// TwinCAT 3 PLC project SaftyPLC
// ProgramVersion: 3.1.4026.13
// libraries:
//   Tc2_Standard, * (Beckhoff Automation GmbH)
//   Tc2_System, * (Beckhoff Automation GmbH)
//   Tc3_Module, * (Beckhoff Automation GmbH)
// project tree:
//   GVLs/ GVL_Safety.TcGVL
//   / PlcTask.TcTTO
//   POUs/ MAIN.TcPOU
// (motion and I/O tree: see PLC project planartrackmovement)
// real-time tasks:
//   TASK XTS Task: cycle T#500us, priority 1, ADS port 350
//   TASK Job Task: cycle default, priority 32
//   TASK MC-Task (MET): cycle T#2ms, priority 3, ADS port 521
//   TASK MC-Task (MPT): cycle T#10ms, priority 8, ADS port 531
//   TASK PlcTask: cycle T#2ms, priority 20, ADS port 351
// variable links:
//   SaftyPLC/SaftyPLC Instance <-> Device 1 (EtherCAT)/Term 1 (EK1200)/Term 13 (EL2912)
//     PlcTask Inputs/GVL_Safety.SaeftyOk <-> StandardInputs/TwinSafeGroup1.SafetyOk_72
//     PlcTask Inputs/GVL_Safety.SafetyInRun <-> StandardInputs/TwinSafeGroup1.SafetyInRun_73
//     PlcTask Outputs/GVL_Safety.Reset <-> StandardOutputs/TwinSafeGroup1.ErrorAcknowledgement_1
//     PlcTask Outputs/GVL_Safety.Run <-> StandardOutputs/TwinSafeGroup1.Run_2
//     PlcTask Outputs/GVL_Safety.Start <-> StandardOutputs/TwinSafeGroup1.STO_75
//   SaftyPLC/SaftyPLC Instance <-> Device 1 (EtherCAT)/Term 1 (EK1200)/Term 2 (EL1809)
//     PlcTask Inputs/GVL_Safety.HWReset <-> Channel 16/Input
//     PlcTask Inputs/GVL_Safety.HWStart <-> Channel 14/Input
//     PlcTask Inputs/GVL_Safety.HWStop <-> Channel 15/Input
//   SaftyPLC/SaftyPLC Instance <-> Device 1 (EtherCAT)/Term 1 (EK1200)/Term 4 (EL2809)
//     PlcTask Outputs/MAIN.xRequestReset <-> Channel 16/Output
//   SaftyPLC/SaftyPLC Instance <-> Device 4 (EtherCAT)/Box 50 (AT5100-0100)
//     PlcTask Outputs/GVL_Safety.Reset <-> Module 1 (SAFETY)/SAFETY Standard Outputdata/Standard In Var 1
//     PlcTask Outputs/GVL_Safety.Run <-> Module 1 (SAFETY)/SAFETY Standard Outputdata/Standard In Var 2
//   SaftyPLC/SaftyPLC Instance <-> Device 4 (EtherCAT)/Box 51 (AT5100-0100)
//     PlcTask Outputs/GVL_Safety.Reset <-> Module 1 (SAFETY)/SAFETY Standard Outputdata/Standard In Var 1
//     PlcTask Outputs/GVL_Safety.Run <-> Module 1 (SAFETY)/SAFETY Standard Outputdata/Standard In Var 2
//   SaftyPLC/SaftyPLC Instance <-> Device 4 (EtherCAT)/Box 52 (AT5100-0100)
//     PlcTask Outputs/GVL_Safety.Reset <-> Module 1 (SAFETY)/SAFETY Standard Outputdata/Standard In Var 1
//     PlcTask Outputs/GVL_Safety.Run <-> Module 1 (SAFETY)/SAFETY Standard Outputdata/Standard In Var 2
//   SaftyPLC/SaftyPLC Instance <-> Device 4 (EtherCAT)/Box 53 (AT5100-0100)
//     PlcTask Outputs/GVL_Safety.Reset <-> Module 1 (SAFETY)/SAFETY Standard Outputdata/Standard In Var 1
//     PlcTask Outputs/GVL_Safety.Run <-> Module 1 (SAFETY)/SAFETY Standard Outputdata/Standard In Var 2
//   SaftyPLC/SaftyPLC Instance <-> Device 4 (EtherCAT)/Box 54 (AT5100-0100)
//     PlcTask Outputs/GVL_Safety.Reset <-> Module 1 (SAFETY)/SAFETY Standard Outputdata/Standard In Var 1
//     PlcTask Outputs/GVL_Safety.Run <-> Module 1 (SAFETY)/SAFETY Standard Outputdata/Standard In Var 2
//   SaftyPLC/SaftyPLC Instance <-> Device 4 (EtherCAT)/Box 55 (AT5100-0100)
//     PlcTask Outputs/GVL_Safety.Reset <-> Module 1 (SAFETY)/SAFETY Standard Outputdata/Standard In Var 1
//     PlcTask Outputs/GVL_Safety.Run <-> Module 1 (SAFETY)/SAFETY Standard Outputdata/Standard In Var 2
//   SaftyPLC/SaftyPLC Instance <-> Device 4 (EtherCAT)/Box 56 (AT5100-0100)
//     PlcTask Outputs/GVL_Safety.Reset <-> Module 1 (SAFETY)/SAFETY Standard Outputdata/Standard In Var 1
//     PlcTask Outputs/GVL_Safety.Run <-> Module 1 (SAFETY)/SAFETY Standard Outputdata/Standard In Var 2
//   SaftyPLC/SaftyPLC Instance <-> Device 4 (EtherCAT)/Box 57 (AT5100-0100)
//     PlcTask Outputs/GVL_Safety.Reset <-> Module 1 (SAFETY)/SAFETY Standard Outputdata/Standard In Var 1
//     PlcTask Outputs/GVL_Safety.Run <-> Module 1 (SAFETY)/SAFETY Standard Outputdata/Standard In Var 2
//   SaftyPLC/SaftyPLC Instance <-> Device 4 (EtherCAT)/Box 58 (AT5100-0100)
//     PlcTask Outputs/GVL_Safety.Reset <-> Module 1 (SAFETY)/SAFETY Standard Outputdata/Standard In Var 1
//     PlcTask Outputs/GVL_Safety.Run <-> Module 1 (SAFETY)/SAFETY Standard Outputdata/Standard In Var 2
//   SaftyPLC/SaftyPLC Instance <-> Device 4 (EtherCAT)/Box 59 (AT5100-0100)
//     PlcTask Outputs/GVL_Safety.Reset <-> Module 1 (SAFETY)/SAFETY Standard Outputdata/Standard In Var 1
//     PlcTask Outputs/GVL_Safety.Run <-> Module 1 (SAFETY)/SAFETY Standard Outputdata/Standard In Var 2
//   SaftyPLC/SaftyPLC Instance <-> Device 4 (EtherCAT)/Box 60 (AT5100-0100)
//     PlcTask Outputs/GVL_Safety.Reset <-> Module 1 (SAFETY)/SAFETY Standard Outputdata/Standard In Var 1
//     PlcTask Outputs/GVL_Safety.Run <-> Module 1 (SAFETY)/SAFETY Standard Outputdata/Standard In Var 2
//   SaftyPLC/SaftyPLC Instance <-> Device 4 (EtherCAT)/Box 61 (AT5100-0100)
//     PlcTask Outputs/GVL_Safety.Reset <-> Module 1 (SAFETY)/SAFETY Standard Outputdata/Standard In Var 1
//     PlcTask Outputs/GVL_Safety.Run <-> Module 1 (SAFETY)/SAFETY Standard Outputdata/Standard In Var 2
//   SaftyPLC/SaftyPLC Instance <-> Device 4 (EtherCAT)/Box 62 (AT5100-0100)
//     PlcTask Outputs/GVL_Safety.Reset <-> Module 1 (SAFETY)/SAFETY Standard Outputdata/Standard In Var 1
//     PlcTask Outputs/GVL_Safety.Run <-> Module 1 (SAFETY)/SAFETY Standard Outputdata/Standard In Var 2
//   SaftyPLC/SaftyPLC Instance <-> Device 4 (EtherCAT)/Box 63 (AT5100-0100)
//     PlcTask Outputs/GVL_Safety.Reset <-> Module 1 (SAFETY)/SAFETY Standard Outputdata/Standard In Var 1
//     PlcTask Outputs/GVL_Safety.Run <-> Module 1 (SAFETY)/SAFETY Standard Outputdata/Standard In Var 2
//   SaftyPLC/SaftyPLC Instance <-> Device 4 (EtherCAT)/Box 64 (AT5100-0100)
//     PlcTask Outputs/GVL_Safety.Reset <-> Module 1 (SAFETY)/SAFETY Standard Outputdata/Standard In Var 1
//     PlcTask Outputs/GVL_Safety.Run <-> Module 1 (SAFETY)/SAFETY Standard Outputdata/Standard In Var 2
//   SaftyPLC/SaftyPLC Instance <-> Device 4 (EtherCAT)/Box 65 (AT5100-0100)
//     PlcTask Outputs/GVL_Safety.Reset <-> Module 1 (SAFETY)/SAFETY Standard Outputdata/Standard In Var 1
//     PlcTask Outputs/GVL_Safety.Run <-> Module 1 (SAFETY)/SAFETY Standard Outputdata/Standard In Var 2
//   SaftyPLC/SaftyPLC Instance <-> Device 4 (EtherCAT)/Box 66 (AT5100-0100)
//     PlcTask Outputs/GVL_Safety.Reset <-> Module 1 (SAFETY)/SAFETY Standard Outputdata/Standard In Var 1
//     PlcTask Outputs/GVL_Safety.Run <-> Module 1 (SAFETY)/SAFETY Standard Outputdata/Standard In Var 2
//   SaftyPLC/SaftyPLC Instance <-> Device 4 (EtherCAT)/Box 67 (AT5100-0100)
//     PlcTask Outputs/GVL_Safety.Reset <-> Module 1 (SAFETY)/SAFETY Standard Outputdata/Standard In Var 1
//     PlcTask Outputs/GVL_Safety.Run <-> Module 1 (SAFETY)/SAFETY Standard Outputdata/Standard In Var 2
//   SaftyPLC/SaftyPLC Instance <-> Device 4 (EtherCAT)/Box 68 (AT5100-0100)
//     PlcTask Outputs/GVL_Safety.Reset <-> Module 1 (SAFETY)/SAFETY Standard Outputdata/Standard In Var 1
//     PlcTask Outputs/GVL_Safety.Run <-> Module 1 (SAFETY)/SAFETY Standard Outputdata/Standard In Var 2
//   SaftyPLC/SaftyPLC Instance <-> Device 4 (EtherCAT)/Box 69 (AT5100-0100)
//     PlcTask Outputs/GVL_Safety.Reset <-> Module 1 (SAFETY)/SAFETY Standard Outputdata/Standard In Var 1
//     PlcTask Outputs/GVL_Safety.Run <-> Module 1 (SAFETY)/SAFETY Standard Outputdata/Standard In Var 2
//   SaftyPLC/SaftyPLC Instance <-> Device 4 (EtherCAT)/Box 70 (AT5100-0100)
//     PlcTask Outputs/GVL_Safety.Reset <-> Module 1 (SAFETY)/SAFETY Standard Outputdata/Standard In Var 1
//     PlcTask Outputs/GVL_Safety.Run <-> Module 1 (SAFETY)/SAFETY Standard Outputdata/Standard In Var 2
//   SaftyPLC/SaftyPLC Instance <-> Device 4 (EtherCAT)/Box 71 (AT5100-0100)
//     PlcTask Outputs/GVL_Safety.Reset <-> Module 1 (SAFETY)/SAFETY Standard Outputdata/Standard In Var 1
//     PlcTask Outputs/GVL_Safety.Run <-> Module 1 (SAFETY)/SAFETY Standard Outputdata/Standard In Var 2
//   SaftyPLC/SaftyPLC Instance <-> Device 4 (EtherCAT)/Box 72 (AT5100-0100)
//     PlcTask Outputs/GVL_Safety.Reset <-> Module 1 (SAFETY)/SAFETY Standard Outputdata/Standard In Var 1
//     PlcTask Outputs/GVL_Safety.Run <-> Module 1 (SAFETY)/SAFETY Standard Outputdata/Standard In Var 2
//   SaftyPLC/SaftyPLC Instance <-> Device 4 (EtherCAT)/Box 73 (AT5100-0100)
//     PlcTask Outputs/GVL_Safety.Reset <-> Module 1 (SAFETY)/SAFETY Standard Outputdata/Standard In Var 1
//     PlcTask Outputs/GVL_Safety.Run <-> Module 1 (SAFETY)/SAFETY Standard Outputdata/Standard In Var 2
//   SaftyPLC/SaftyPLC Instance <-> Device 4 (EtherCAT)/Box 74 (AT5100-0100)
//     PlcTask Outputs/GVL_Safety.Reset <-> Module 1 (SAFETY)/SAFETY Standard Outputdata/Standard In Var 1
//     PlcTask Outputs/GVL_Safety.Run <-> Module 1 (SAFETY)/SAFETY Standard Outputdata/Standard In Var 2
//   SaftyPLC/SaftyPLC Instance <-> Device 4 (EtherCAT)/Box 75 (AT5100-0100)
//     PlcTask Outputs/GVL_Safety.Reset <-> Module 1 (SAFETY)/SAFETY Standard Outputdata/Standard In Var 1
//     PlcTask Outputs/GVL_Safety.Run <-> Module 1 (SAFETY)/SAFETY Standard Outputdata/Standard In Var 2
//   SaftyPLC/SaftyPLC Instance <-> Device 4 (EtherCAT)/Box 76 (AT5100-0100)
//     PlcTask Outputs/GVL_Safety.Reset <-> Module 1 (SAFETY)/SAFETY Standard Outputdata/Standard In Var 1
//     PlcTask Outputs/GVL_Safety.Run <-> Module 1 (SAFETY)/SAFETY Standard Outputdata/Standard In Var 2
//   SaftyPLC/SaftyPLC Instance <-> Device 4 (EtherCAT)/Box 77 (AT5100-0100)
//     PlcTask Outputs/GVL_Safety.Reset <-> Module 1 (SAFETY)/SAFETY Standard Outputdata/Standard In Var 1
//     PlcTask Outputs/GVL_Safety.Run <-> Module 1 (SAFETY)/SAFETY Standard Outputdata/Standard In Var 2
//   SaftyPLC/SaftyPLC Instance <-> Device 4 (EtherCAT)/Box 78 (AT5100-0100)
//     PlcTask Outputs/GVL_Safety.Reset <-> Module 1 (SAFETY)/SAFETY Standard Outputdata/Standard In Var 1
//     PlcTask Outputs/GVL_Safety.Run <-> Module 1 (SAFETY)/SAFETY Standard Outputdata/Standard In Var 2
//   SaftyPLC/SaftyPLC Instance <-> Device 4 (EtherCAT)/Box 79 (AT5100-0100)
//     PlcTask Outputs/GVL_Safety.Reset <-> Module 1 (SAFETY)/SAFETY Standard Outputdata/Standard In Var 1
//     PlcTask Outputs/GVL_Safety.Run <-> Module 1 (SAFETY)/SAFETY Standard Outputdata/Standard In Var 2
//   SaftyPLC/SaftyPLC Instance <-> Device 4 (EtherCAT)/Box 80 (AT5100-0100)
//     PlcTask Outputs/GVL_Safety.Reset <-> Module 1 (SAFETY)/SAFETY Standard Outputdata/Standard In Var 1
//     PlcTask Outputs/GVL_Safety.Run <-> Module 1 (SAFETY)/SAFETY Standard Outputdata/Standard In Var 2
//   SaftyPLC/SaftyPLC Instance <-> Device 4 (EtherCAT)/Box 81 (AT5100-0100)
//     PlcTask Outputs/GVL_Safety.Reset <-> Module 1 (SAFETY)/SAFETY Standard Outputdata/Standard In Var 1
//     PlcTask Outputs/GVL_Safety.Run <-> Module 1 (SAFETY)/SAFETY Standard Outputdata/Standard In Var 2
//   SaftyPLC/SaftyPLC Instance <-> Device 8 (EtherCAT)/Box 18 (AT5100-0100)
//     PlcTask Outputs/GVL_Safety.Reset <-> Module 1 (SAFETY)/SAFETY Standard Outputdata/Standard In Var 1
//     PlcTask Outputs/GVL_Safety.Run <-> Module 1 (SAFETY)/SAFETY Standard Outputdata/Standard In Var 2
//   SaftyPLC/SaftyPLC Instance <-> Device 8 (EtherCAT)/Box 19 (AT5100-0100)
//     PlcTask Outputs/GVL_Safety.Reset <-> Module 1 (SAFETY)/SAFETY Standard Outputdata/Standard In Var 1
//     PlcTask Outputs/GVL_Safety.Run <-> Module 1 (SAFETY)/SAFETY Standard Outputdata/Standard In Var 2
//   SaftyPLC/SaftyPLC Instance <-> Device 8 (EtherCAT)/Box 20 (AT5100-0100)
//     PlcTask Outputs/GVL_Safety.Reset <-> Module 1 (SAFETY)/SAFETY Standard Outputdata/Standard In Var 1
//     PlcTask Outputs/GVL_Safety.Run <-> Module 1 (SAFETY)/SAFETY Standard Outputdata/Standard In Var 2
//   SaftyPLC/SaftyPLC Instance <-> Device 8 (EtherCAT)/Box 21 (AT5100-0100)
//     PlcTask Outputs/GVL_Safety.Reset <-> Module 1 (SAFETY)/SAFETY Standard Outputdata/Standard In Var 1
//     PlcTask Outputs/GVL_Safety.Run <-> Module 1 (SAFETY)/SAFETY Standard Outputdata/Standard In Var 2
//   SaftyPLC/SaftyPLC Instance <-> Device 8 (EtherCAT)/Box 22 (AT5100-0100)
//     PlcTask Outputs/GVL_Safety.Reset <-> Module 1 (SAFETY)/SAFETY Standard Outputdata/Standard In Var 1
//     PlcTask Outputs/GVL_Safety.Run <-> Module 1 (SAFETY)/SAFETY Standard Outputdata/Standard In Var 2
//   SaftyPLC/SaftyPLC Instance <-> Device 8 (EtherCAT)/Box 23 (AT5100-0100)
//     PlcTask Outputs/GVL_Safety.Reset <-> Module 1 (SAFETY)/SAFETY Standard Outputdata/Standard In Var 1
//     PlcTask Outputs/GVL_Safety.Run <-> Module 1 (SAFETY)/SAFETY Standard Outputdata/Standard In Var 2
//   SaftyPLC/SaftyPLC Instance <-> Device 8 (EtherCAT)/Box 24 (AT5100-0100)
//     PlcTask Outputs/GVL_Safety.Reset <-> Module 1 (SAFETY)/SAFETY Standard Outputdata/Standard In Var 1
//     PlcTask Outputs/GVL_Safety.Run <-> Module 1 (SAFETY)/SAFETY Standard Outputdata/Standard In Var 2
//   SaftyPLC/SaftyPLC Instance <-> Device 8 (EtherCAT)/Box 25 (AT5100-0100)
//     PlcTask Outputs/GVL_Safety.Reset <-> Module 1 (SAFETY)/SAFETY Standard Outputdata/Standard In Var 1
//     PlcTask Outputs/GVL_Safety.Run <-> Module 1 (SAFETY)/SAFETY Standard Outputdata/Standard In Var 2
//   SaftyPLC/SaftyPLC Instance <-> Device 8 (EtherCAT)/Box 26 (AT5100-0100)
//     PlcTask Outputs/GVL_Safety.Reset <-> Module 1 (SAFETY)/SAFETY Standard Outputdata/Standard In Var 1
//     PlcTask Outputs/GVL_Safety.Run <-> Module 1 (SAFETY)/SAFETY Standard Outputdata/Standard In Var 2
//   SaftyPLC/SaftyPLC Instance <-> Device 8 (EtherCAT)/Box 27 (AT5100-0100)
//     PlcTask Outputs/GVL_Safety.Reset <-> Module 1 (SAFETY)/SAFETY Standard Outputdata/Standard In Var 1
//     PlcTask Outputs/GVL_Safety.Run <-> Module 1 (SAFETY)/SAFETY Standard Outputdata/Standard In Var 2
//   SaftyPLC/SaftyPLC Instance <-> Device 8 (EtherCAT)/Box 28 (AT5100-0100)
//     PlcTask Outputs/GVL_Safety.Reset <-> Module 1 (SAFETY)/SAFETY Standard Outputdata/Standard In Var 1
//     PlcTask Outputs/GVL_Safety.Run <-> Module 1 (SAFETY)/SAFETY Standard Outputdata/Standard In Var 2
//   SaftyPLC/SaftyPLC Instance <-> Device 8 (EtherCAT)/Box 29 (AT5100-0100)
//     PlcTask Outputs/GVL_Safety.Reset <-> Module 1 (SAFETY)/SAFETY Standard Outputdata/Standard In Var 1
//     PlcTask Outputs/GVL_Safety.Run <-> Module 1 (SAFETY)/SAFETY Standard Outputdata/Standard In Var 2
//   SaftyPLC/SaftyPLC Instance <-> Device 8 (EtherCAT)/Box 30 (AT5100-0100)
//     PlcTask Outputs/GVL_Safety.Reset <-> Module 1 (SAFETY)/SAFETY Standard Outputdata/Standard In Var 1
//     PlcTask Outputs/GVL_Safety.Run <-> Module 1 (SAFETY)/SAFETY Standard Outputdata/Standard In Var 2
//   SaftyPLC/SaftyPLC Instance <-> Device 8 (EtherCAT)/Box 31 (AT5100-0100)
//     PlcTask Outputs/GVL_Safety.Reset <-> Module 1 (SAFETY)/SAFETY Standard Outputdata/Standard In Var 1
//     PlcTask Outputs/GVL_Safety.Run <-> Module 1 (SAFETY)/SAFETY Standard Outputdata/Standard In Var 2
//   SaftyPLC/SaftyPLC Instance <-> Device 8 (EtherCAT)/Box 32 (AT5100-0100)
//     PlcTask Outputs/GVL_Safety.Reset <-> Module 1 (SAFETY)/SAFETY Standard Outputdata/Standard In Var 1
//     PlcTask Outputs/GVL_Safety.Run <-> Module 1 (SAFETY)/SAFETY Standard Outputdata/Standard In Var 2
//   SaftyPLC/SaftyPLC Instance <-> Device 8 (EtherCAT)/Box 33 (AT5100-0100)
//     PlcTask Outputs/GVL_Safety.Reset <-> Module 1 (SAFETY)/SAFETY Standard Outputdata/Standard In Var 1
//     PlcTask Outputs/GVL_Safety.Run <-> Module 1 (SAFETY)/SAFETY Standard Outputdata/Standard In Var 2
//   SaftyPLC/SaftyPLC Instance <-> Device 8 (EtherCAT)/Box 34 (AT5100-0100)
//     PlcTask Outputs/GVL_Safety.Reset <-> Module 1 (SAFETY)/SAFETY Standard Outputdata/Standard In Var 1
//     PlcTask Outputs/GVL_Safety.Run <-> Module 1 (SAFETY)/SAFETY Standard Outputdata/Standard In Var 2
//   SaftyPLC/SaftyPLC Instance <-> Device 8 (EtherCAT)/Box 35 (AT5100-0100)
//     PlcTask Outputs/GVL_Safety.Reset <-> Module 1 (SAFETY)/SAFETY Standard Outputdata/Standard In Var 1
//     PlcTask Outputs/GVL_Safety.Run <-> Module 1 (SAFETY)/SAFETY Standard Outputdata/Standard In Var 2
//   SaftyPLC/SaftyPLC Instance <-> Device 8 (EtherCAT)/Box 36 (AT5100-0100)
//     PlcTask Outputs/GVL_Safety.Reset <-> Module 1 (SAFETY)/SAFETY Standard Outputdata/Standard In Var 1
//     PlcTask Outputs/GVL_Safety.Run <-> Module 1 (SAFETY)/SAFETY Standard Outputdata/Standard In Var 2
//   SaftyPLC/SaftyPLC Instance <-> Device 8 (EtherCAT)/Box 37 (AT5100-0100)
//     PlcTask Outputs/GVL_Safety.Reset <-> Module 1 (SAFETY)/SAFETY Standard Outputdata/Standard In Var 1
//     PlcTask Outputs/GVL_Safety.Run <-> Module 1 (SAFETY)/SAFETY Standard Outputdata/Standard In Var 2
//   SaftyPLC/SaftyPLC Instance <-> Device 8 (EtherCAT)/Box 38 (AT5100-0100)
//     PlcTask Outputs/GVL_Safety.Reset <-> Module 1 (SAFETY)/SAFETY Standard Outputdata/Standard In Var 1
//     PlcTask Outputs/GVL_Safety.Run <-> Module 1 (SAFETY)/SAFETY Standard Outputdata/Standard In Var 2
//   SaftyPLC/SaftyPLC Instance <-> Device 8 (EtherCAT)/Box 39 (AT5100-0100)
//     PlcTask Outputs/GVL_Safety.Reset <-> Module 1 (SAFETY)/SAFETY Standard Outputdata/Standard In Var 1
//     PlcTask Outputs/GVL_Safety.Run <-> Module 1 (SAFETY)/SAFETY Standard Outputdata/Standard In Var 2
//   SaftyPLC/SaftyPLC Instance <-> Device 8 (EtherCAT)/Box 40 (AT5100-0100)
//     PlcTask Outputs/GVL_Safety.Reset <-> Module 1 (SAFETY)/SAFETY Standard Outputdata/Standard In Var 1
//     PlcTask Outputs/GVL_Safety.Run <-> Module 1 (SAFETY)/SAFETY Standard Outputdata/Standard In Var 2
//   SaftyPLC/SaftyPLC Instance <-> Device 8 (EtherCAT)/Box 41 (AT5100-0100)
//     PlcTask Outputs/GVL_Safety.Reset <-> Module 1 (SAFETY)/SAFETY Standard Outputdata/Standard In Var 1
//     PlcTask Outputs/GVL_Safety.Run <-> Module 1 (SAFETY)/SAFETY Standard Outputdata/Standard In Var 2
//   SaftyPLC/SaftyPLC Instance <-> Device 8 (EtherCAT)/Box 42 (AT5100-0100)
//     PlcTask Outputs/GVL_Safety.Reset <-> Module 1 (SAFETY)/SAFETY Standard Outputdata/Standard In Var 1
//     PlcTask Outputs/GVL_Safety.Run <-> Module 1 (SAFETY)/SAFETY Standard Outputdata/Standard In Var 2
//   SaftyPLC/SaftyPLC Instance <-> Device 8 (EtherCAT)/Box 43 (AT5100-0100)
//     PlcTask Outputs/GVL_Safety.Reset <-> Module 1 (SAFETY)/SAFETY Standard Outputdata/Standard In Var 1
//     PlcTask Outputs/GVL_Safety.Run <-> Module 1 (SAFETY)/SAFETY Standard Outputdata/Standard In Var 2
//   SaftyPLC/SaftyPLC Instance <-> Device 8 (EtherCAT)/Box 44 (AT5100-0100)
//     PlcTask Outputs/GVL_Safety.Reset <-> Module 1 (SAFETY)/SAFETY Standard Outputdata/Standard In Var 1
//     PlcTask Outputs/GVL_Safety.Run <-> Module 1 (SAFETY)/SAFETY Standard Outputdata/Standard In Var 2
//   SaftyPLC/SaftyPLC Instance <-> Device 8 (EtherCAT)/Box 45 (AT5100-0100)
//     PlcTask Outputs/GVL_Safety.Reset <-> Module 1 (SAFETY)/SAFETY Standard Outputdata/Standard In Var 1
//     PlcTask Outputs/GVL_Safety.Run <-> Module 1 (SAFETY)/SAFETY Standard Outputdata/Standard In Var 2
//   SaftyPLC/SaftyPLC Instance <-> Device 8 (EtherCAT)/Box 46 (AT5100-0100)
//     PlcTask Outputs/GVL_Safety.Reset <-> Module 1 (SAFETY)/SAFETY Standard Outputdata/Standard In Var 1
//     PlcTask Outputs/GVL_Safety.Run <-> Module 1 (SAFETY)/SAFETY Standard Outputdata/Standard In Var 2
//   SaftyPLC/SaftyPLC Instance <-> Device 8 (EtherCAT)/Box 47 (AT5100-0100)
//     PlcTask Outputs/GVL_Safety.Reset <-> Module 1 (SAFETY)/SAFETY Standard Outputdata/Standard In Var 1
//     PlcTask Outputs/GVL_Safety.Run <-> Module 1 (SAFETY)/SAFETY Standard Outputdata/Standard In Var 2
//   SaftyPLC/SaftyPLC Instance <-> Device 8 (EtherCAT)/Box 48 (AT5100-0100)
//     PlcTask Outputs/GVL_Safety.Reset <-> Module 1 (SAFETY)/SAFETY Standard Outputdata/Standard In Var 1
//     PlcTask Outputs/GVL_Safety.Run <-> Module 1 (SAFETY)/SAFETY Standard Outputdata/Standard In Var 2
//   SaftyPLC/SaftyPLC Instance <-> Device 8 (EtherCAT)/Box 49 (AT5100-0100)
//     PlcTask Outputs/GVL_Safety.Reset <-> Module 1 (SAFETY)/SAFETY Standard Outputdata/Standard In Var 1
//     PlcTask Outputs/GVL_Safety.Run <-> Module 1 (SAFETY)/SAFETY Standard Outputdata/Standard In Var 2

CONFIGURATION SaftyPLC
    RESOURCE PLC ON TwinCAT3
        TASK PlcTask(INTERVAL := T#2ms, PRIORITY := 20);
        PROGRAM MAIN WITH PlcTask : MAIN;
    END_RESOURCE
END_CONFIGURATION

// ---- GVLs/GVL_Safety.TcGVL
{attribute 'qualified_only'}
VAR_GLOBAL
	Run			AT%Q* : BOOL := TRUE;
	Start		AT%Q* : BOOL := TRUE;
	Reset		AT%Q* : BOOL;
	
	SafetyInRun	AT%I* : BOOL;
	SaeftyOk 	AT%I* : BOOL;
	
	HWStart		AT%I* : BOOL;
	HWStop		AT%I* : BOOL;
	HWReset		AT%I* : BOOL;
	
	HWerror		AT%Q* : BOOL;
	HWSafetyOk	AT%Q* : BOOL;
	
END_VAR

// ---- POUs/MAIN.TcPOU
PROGRAM MAIN
VAR
	nCase 					: INT;
	
	xRequestReset 	AT%Q* 	: BOOL;
	xError 				 	: BOOL;
		

	rTrigSwitchon 		  	: R_trig;
	fTrigSwitchOff		  	: F_trig;
	Chargtimer 				: ton;
	
	SwitchOn				: BOOL;
	SoftReset 				: bool;

END_VAR



IF GVL_Safety.HWStart THEN
	GVL_Safety.Run  := TRUE;
	GVL_Safety.Start := TRUE;
END_IF

IF  NOT GVL_Safety.HWStop THEN
	GVL_Safety.Run  := FALSE;
	GVL_Safety.Start := FALSE;
END_IF
		


IF gvl_safety.SaeftyOk THEN
	gvl_safety.HWSafetyOk := TRUE;
ELSE	
	gvl_safety.HWSafetyOk := FALSE;
END_IF

IF NOT gvl_safety.SafetyInRun THEN
	gvl_safety.HWerror := TRUE;
ELSE	
	gvl_safety.HWerror := FALSE;
END_IF

xError := NOT gvl_safety.SafetyInRun AND NOT gvl_safety.HWSafetyOk AND GVL_Safety.Run AND GVL_Safety.Start;

xRequestReset	:= NOT GVL_Safety.SaeftyOk;

IF GVL_safety.hwReset OR SoftReset  THEN
	GVL_Safety.Reset := TRUE;
ELSE 	
	GVL_Safety.Reset := FALSE;
END_IF

END_PROGRAM
